Omron CX-Programmer project NewProject (CX-Programmer 9.61)

# PLC NewPLC1: CJ2M CPU31
I/O table (CPU CJ2M-CPU31): rack 0 slot 0 CJ1W-AD041-V1; rack 0 slot 1 CJ1W-ID211; rack 0 slot 2 CJ1W-OD211; rack 0 slot 3 CJ1W-DA041; rack 0 slot 11 CJ2M-EIP21

## Global symbols (name address type ; comment)
0.00 BOOL  ; PB_EMERGENCY STOP
0.01 BOOL  ; PB_MAN/AUTO
0.02 BOOL  ; PB_START
0.03 BOOL  ; PB_STOP
0.04 BOOL  ; PB_RESET
0.05 BOOL  ; PART SENSOR
0.06 BOOL  ; JIG IAI RIGHT END
0.07 BOOL  ; JIG IAI LEFT END
0.08 BOOL  ; JIG IAI ALARM
0.09 BOOL  ; INKJET IAI UP END
0.10 BOOL  ; INKJET IAI DOWN END
0.11 BOOL  ; INKJET IAI ALARM
0.12 BOOL  ; INKJET ERROR
0.13 BOOL  ; INKJET REFILL WARNING
0.14 BOOL  ; INKJET READY
0.15 BOOL  ; SPARE
1519.11 BOOL  ; Sequence end complete
1519.15 BOOL  ; Protocol Macro Executing
1.00 BOOL  ; LAMP PB_START
1.01 BOOL  ; JIG IAI RIGHT
1.02 BOOL  ; JIG IAI LEFT
1.03 BOOL  ; INKJET IAI UP
1.04 BOOL  ; INKJET IAI DOWN
1.05 BOOL  ; ALL IAI RESET ALARM
1.06 BOOL  ; BUZZER
1.07 BOOL  ; TWL YELLOW
1.08 BOOL  ; TWL GREEN
1.09 BOOL  ; TWL RED
1.10 BOOL  ; GREEN OK TWL
1.11 BOOL  ; RED NG TWL
2.00 BOOL  ; INKJET X4 IN1
2.01 BOOL  ; INKJET X4 IN2
2.02 BOOL  ; INKJET X4 IN3
2.03 BOOL  ; INKJET X4 JOB0
2.04 BOOL  ; INKJET X4 JOB1
2.05 BOOL  ; INKJET X4 JOB2
2.06 BOOL  ; INKJET X4 JOB3
2.07 BOOL  ; INKJET X4 JOB4
2.08 BOOL  ; INKJET X4 JOB5
2.09 BOOL  ; INKJET X4 JOB6
2.10 BOOL  ; INKJET X4 JOB7
2.11 BOOL  ; PRINT GO
3.00 BOOL  ; SOL ROTATE WORKPIECE ADV.
3.01 BOOL  ; SOL ROTATE WORKPIECE RET.
3.02 BOOL  ; SOL EJECTOR WORK NG ADV.
3.03 BOOL  ; SOL EJECTOR WORK NG RET.
3.04 BOOL  ; SOL CUT-OFF ADV.
3.05 BOOL  ; SOL CUT-OFF RET.
3.06 BOOL  ; SOL HOPPER ADV.
3.07 BOOL  ; SOL HOPPER RET.
3.08 BOOL  ; + JOB SELECT 0 (INKJET)
3.09 BOOL  ; + JOB SELECT 1 (INKJET)
3.10 BOOL  ; + JOB SELECT 2 (INKJET)
3.11 BOOL  ; + JOB SELECT 3 (INKJET)
3.12 BOOL  ; + JOB SELECT 4 (INKJET)
3.13 BOOL  ; + JOB SELECT 5 (INKJET)
3.14 BOOL  ; + JOB SELECT 6 (INKJET)
3.15 BOOL  ; + JOB SELECT 7 (INKJET)
40.09 BOOL  ; WARNING PRINT AGAIN
500.00 BOOL  ; SR-1000_PLC timming area
700.02 BOOL  ; TS170 TP WRITE DATA
750.05 BOOL  ; READING OK SV
850.00 BOOL  ; B-15 MANUAL HOME SELECT
950.00 BOOL  ; DTAT LOG INPUT
A202.07 BOOL  ; Com port Enable
A280.03 BOOL  ; COMPLETE
A280.05 BOOL  ; SERVO HOME
D0 CHANNEL  ; SCREEN CHANGE
D1 CHANNEL  ; 50.0% vari to G3PW
D100 CHANNEL  ; COUNTER PART
D1000 CHANNEL  ; MODEL NAME RUNNING
D102 CHANNEL  ; COUNTER PART NG
D1030 CHANNEL  ; PARM Q'TY BOX
D1050.00 BOOL  ; + JOB SELECT 0 (PLC PARAMETER)
D1050.01 BOOL  ; + JOB SELECT 1 (PLC PARAMETER)
D1050.02 BOOL  ; + JOB SELECT 2 (PLC PARAMETER)
D1050.03 BOOL  ; + JOB SELECT 3 (PLC PARAMETER)
D1050.04 BOOL  ; + JOB SELECT 4 (PLC PARAMETER)
D1050.05 BOOL  ; + JOB SELECT 5 (PLC PARAMETER)
D1050.06 BOOL  ; + JOB SELECT 6 (PLC PARAMETER)
D1050.07 BOOL  ; + JOB SELECT 7 (PLC PARAMETER)
D107 CHANNEL  ; DELAY BEFORE ADV
D108 CHANNEL  ; STATE OK NG
D110 CHANNEL  ; CYCLE TIME
D112 CHANNEL  ; CYCLE TIME
D114 CHANNEL  ; BARCODE TRIG DELAY
D116 CHANNEL  ; EJECTOR DELAY
D15 CHANNEL  ; TSC SET DELAY START
D19 CHANNEL  ; STATUS DISPLAY
D1900 CHANNEL  ; MODEL 1Y  2Wh 3BL 4Grey
D196 CHANNEL  ; CHANGE BOX NUMBER.
D1990 CHANNEL  ; MODEL NUMBER
D200 CHANNEL  ; FLT OKPART COUNT
D2000 CHANNEL  ; SCANNER DATA COMPARE
D210 CHANNEL  ; FEEDRATE COUNT
D220 CHANNEL  ; Password
D230 CHANNEL  ; FEERATE TSC.
D232 CHANNEL  ; OK PART COUNT
D234 CHANNEL  ; CHANGE BOX COUNT.
D236 CHANNEL  ; AGV SHOT TARGET
D240 CHANNEL  ; PART/SHOT COUNT
D244 CHANNEL  ; NG COUNT ALARM
D246 CHANNEL  ; NG COUNT TARGET
D248 CHANNEL  ; TIME OUT ALARM
D2500 CHANNEL  ; Cear Events Password
D260 CHANNEL  ; SHOT COUNT
D30000 CHANNEL  ; DATALOGGING
D3001.01 BOOL  ; ok
D3001.02 BOOL  ; ng
D3002.00 BOOL  ; Fins Ok
D3002.01 BOOL  ; Cam ok
D400 CHANNEL  ; DATA READ FROM SCANNER
D4990 CHANNEL  ; MODEL NUMBER
D4992 CHANNEL  ; MODEL NUMBER -1
D4994 CHANNEL  ; MODEL NUMBER -1*200
D4996 CHANNEL  ; ADDRESS START
D5000 CHANNEL  ; PARAMETER MODEL NAME
D504 CHANNEL  ; DATA READ FROM SCANNER
D600 CHANNEL  ; DATA READ FROM SCANNER IN PAGE32
D810 CHANNEL  ; POSITION FORM SELECT
D900 CHANNEL  ; AUTO DATA READ FROMSCANNER
H0.01 BOOL  ; MANUAL SELECT
H0.02 BOOL  ; AUTO SELECT
H100.00 BOOL  ; Z SELECT DIRECTION
H10.00 BOOL  ; STATE SIZE 80 USED
H10.01 BOOL  ; STATE SIZE 100 USE
H10.02 BOOL  ; STATE SIZE 150 USED
H11.00 BOOL  ; SIZE 80 USED
H11.01 BOOL  ; SIZE 100 USED
H11.02 BOOL  ; SIZE 150 USED
H12 CHANNEL  ; CHANGE PIC MODEL
H25.00 BOOL  ; USE COLOR DETECT
H420.15 BOOL  ; ALL FAULT(OFF)
H7.00 BOOL  ; SWITCH SELECTED
H7.01 BOOL  ; SENSOR SELECTED
H8.00 BOOL  ; BARCODE DISABLE
H8.01 BOOL  ; USE/UN USE INKJET
H8.02 BOOL  ; CHANGE BOX.
T0000 BOOL  ; BEFORE FLIP CYL. ADV
T0001 BOOL  ; AFTER FLIP CYL. ADV
T0008 BOOL  ; SS MODE MANUAL/AUTO [0.04] On
T0009 BOOL  ; SS MODE MANUAL/AUTO [0.04] Off
T0020 BOOL  ; DELAY START FROM SENSOR
T0021 BOOL  ; POWER ON TIME
T0050 BOOL  ; DELAY START BOWL
T0051 BOOL  ; DELAY PRINT GO
T0055 BOOL  ; NG BUFFER1 RUNNING
T0056 BOOL  ; NG BUFFER2 RUNNING
T0070 BOOL  ; EJECTOR TRIG BUFFER1
T0073 BOOL  ; EJECTOR TRIG BUFFER2
T0081 BOOL  ; EJECTOR RIGHT ALM.
T0082 BOOL  ; BUFFER BOX ADV. ALM.
T0083 BOOL  ; BUFFER BOX RET ALM.
T0092 BOOL  ; TIME OFF NG
T0093 BOOL  ; TIME OUT
T0098 BOOL  ; READ DONE
T0100 BOOL  ; AS EJECTOR WORK NG ADV. [1.02] On
T0101 BOOL  ; AS EJECTOR WORK NG RET. [1.03] On
T0102 BOOL  ; NG BUFFER3 RUNNING
T0103 BOOL  ; AS CUT-OFF RET. [1.05] On
T0104 BOOL  ; AS HOPPER ADV. [1.06] On
T0105 BOOL  ; AS HOPPER RET. [1.07] On
T0110 BOOL  ; AS ROTATE WORK PIECE ADV. [1.00] On
T0111 BOOL  ; AS ROTATE WORK PIECE RET. [1.01] On
T0152 BOOL  ; PH CHECK WORK EJECTOR  [1.10] On
T0153 BOOL  ; PH CHECK WORK EJECTOR  [1.10] Off
T0155 BOOL  ; PH CHECK WORK COUNTER [1.11] Off
T1002 BOOL  ; TIMER PREPARE DATA
T2000 BOOL  ; TIMER MODEL NAME SET
W0.00 BOOL  ; EMERGENCY STOP PB.
W0.01 BOOL  ; MANUAL MODE
W0.02 BOOL  ; AUTO MODE
W0.03 BOOL  ; MANUAL MODE PB. TSC.
W0.04 BOOL  ; AUTO MODE PB. TSC.
W0.10 BOOL  ; SET FLIP CYL ADV.
W100.00 BOOL  ; PB_EMERGENCY STOP
W100.01 BOOL  ; PB_MAN/AUTO
W100.02 BOOL  ; PB_START
W100.03 BOOL  ; PB_STOP
W100.04 BOOL  ; PB_RESET
W100.05 BOOL  ; PART SENSOR
W100.06 BOOL  ; JIG IAI RIGHT END
W100.07 BOOL  ; JIG IAI LEFT END
W100.08 BOOL  ; JIG IAI ALARM
W100.09 BOOL  ; INKJET IAI UP END
W100.10 BOOL  ; INKJET IAI DOWN END
W100.11 BOOL  ; INKJET IAI ALARM
W100.12 BOOL  ; INKJET ERROR
W100.13 BOOL  ; INKJET REFILL WARNING
W100.14 BOOL  ; INKJET READY
W100.15 BOOL  ; SPARE
W101.00 BOOL  ; LAMP PB_START
W101.01 BOOL  ; JIG IAI RIGHT
W101.02 BOOL  ; JIG IAI LEFT
W101.03 BOOL  ; INKJET IAI UP
W101.04 BOOL  ; INKJET IAI DOWN
W101.05 BOOL  ; ALL IAI RESET ALARM
W101.06 BOOL  ; INKJET PRINT GO
W101.07 BOOL  ; INKJET X4 IN1
W101.08 BOOL  ; INKJET X4 IN2
W101.09 BOOL  ; INKJET X4 IN2
W101.10 BOOL  ; INKJET X4 JOB0
W101.11 BOOL  ; INKJET X4 JOB1
W101.12 BOOL  ; INKJET X4 JOB2
W101.13 BOOL  ; TWL YELLOW
W101.14 BOOL  ; TWL GREEN
W101.15 BOOL  ; TWL RED
W102.00 BOOL  ; GREEN OK TWL
W102.01 BOOL  ; RED NG TWL
W10.00 BOOL  ; A/JIG IAI RIGHT
W10.01 BOOL  ; A/JIG IAI LEFT
W10.02 BOOL  ; A/INKJET IAI UP
W10.03 BOOL  ; A/INKJET IAI DOWN
W10.04 BOOL  ; A/CONVEYOR START
W10.05 BOOL  ; A/BOWL START
W10.06 BOOL  ; A/PRINT GO
W10.07 BOOL  ; NG BUFFER1
W10.08 BOOL  ; NG BUFFER2
W10.09 BOOL  ; SET NG BUFFER1
W10.10 BOOL  ; SET NG BUFFER2
W10.11 BOOL  ; SET NG BUFFER3
W10.12 BOOL  ; NG BUFFER3
W10.13 BOOL  ; A/SHOT TRIG TO AGV
W10.15 BOOL  ; HOME
W11.00 BOOL  ; EJECTOR RUNNING
W11.01 BOOL  ; CALL JOB 0
W11.02 BOOL  ; CALL JOB 1
W11.03 BOOL  ; CALL JOB 2
W13.00 BOOL  ; CALL JOB 0
W13.01 BOOL  ; CALL JOB 1
W13.02 BOOL  ; CALL JOB 2
W15.00 BOOL  ; BIT TRIG SHOT
W15.01 BOOL  ; AGV LOADING START COUNT BUFFER
W1.00 BOOL  ; start communication
W1.01 BOOL  ; CYCLE START
W1.02 BOOL  ; RETURN DONE
W1.03 BOOL  ; MACHINE READY
W1.04 BOOL  ; A/PRINT GO(DOWN)
W1.05 BOOL  ; A/PRINT GO(UP)
W1.13 BOOL  ; TEST LAMP
W200.11 BOOL  ; AUTO RUNNING
W202.10 BOOL  ; BARCODE CHECK OK
W202.11 BOOL  ; BARCODE CHECK NG
W204.02 BOOL  ; EJECT WORK RUNNING
W20.00 BOOL  ; Delay Check Barcode
W21.00 BOOL  ; ROBOT STOP
W25.02 BOOL  ; FLAG TO DECRETE NG
W26.03 BOOL  ; GREEN
W26.05 BOOL  ; RED
W300.00 BOOL  ; TRIG COLOR DETECT
W300.01 BOOL  ; FINS OK
W300.02 BOOL  ; CAM CONNECT
W300.03 BOOL  ; DETECT OK
W300.04 BOOL  ; DETECT NG
W302.00 BOOL  ; RECORD Y
W302.01 BOOL  ; RECORD WH
W303.00 BOOL  ; MAN. READ COLOR
W304.00 BOOL  ; WARNING CORLOR DETECTION
W305.00 BOOL  ; FIRST START CHECK COLOR
W30.00 BOOL  ; TRIG HMI MACRO 00
W30.01 BOOL  ; TRIG MACRO
W30.02 BOOL  ; TRIG MACRO AUTO PAGE
W345.00 BOOL  ; TS069 PB CLEAR BOX
W345.01 BOOL  ; TSC CLEAR POPUP
W345.02 BOOL  ; ENABLE JUDGMENT
W35 CHANNEL  ; INDIREC SCR AUTO PAGE
W350.00 BOOL  ; TSPL EJECTOR WORK NG ADV.
W350.01 BOOL  ; TSPL EJECTOR WORK NG RET.
W350.02 BOOL  ; TSPL CUT-OFF ADV.
W350.03 BOOL  ; TSPL CUT-OFF RET.
W350.04 BOOL  ; TSPL HOPPER ADV.
W350.05 BOOL  ; TSPL HOPPER RET.
W350.07 BOOL  ; TS PL SCANNER TRIG
W350.08 BOOL  ; TSPL MOTOR CONVEYOR ON
W350.09 BOOL  ; TSPL MOTOR CONVEYOR OFF
W350.10 BOOL  ; TSPL HOPPER BOWL FEEDER ON
W350.11 BOOL  ; TSPL HOPPER BOWL FEEDER OFF
W350.12 BOOL  ; TSPL BOWL FEEDER ON
W350.13 BOOL  ; TSPL BOWL FEEDER OFF
W350.14 BOOL  ; TSPL LINEAR BOWL FEEDER ON
W350.15 BOOL  ; TSPL LINEAR BOWL FEEDER OFF
W351.00 BOOL  ; TS PL ROTATE WORK PIECE ADV.
W351.01 BOOL  ; TS PL ROTATE WORK PIECE RET.
W36 CHANNEL  ; 400X250 INDIRECT SCR AUTO PAGE
W39.09 BOOL  ; ALL ALARM
W39.10 BOOL  ; ALARM
W401 CHANNEL  ; CURRENT SCREEN
W402 CHANNEL  ; CHANGE SCREEN
W40.01 BOOL  ; EMERGENCY STOP
W40.02 BOOL  ; DEVICES NOT HOME
W40.03 BOOL  ; PLC ERROR
W40.04 BOOL  ; PLC LOW BATTERY
W40.05 BOOL  ; JIG IAI ALARM
W40.06 BOOL  ; INKJET IAI ALARM
W40.07 BOOL  ; INKJET ERROR
W40.08 BOOL  ; INKJET REFILL WARNING
W40.09 BOOL  ; FLIP ROD RET. ALM
W40.10 BOOL  ; NG COUNT ALM.
W40.11 BOOL  ; OVER CYCLE TIME ALM.
W40.12 BOOL  ; DOOR OPENED
W40.13 BOOL  ; PART SENSOR ALM.
W40.14 BOOL  ; EJECTOR SENSOR ALM.
W40.15 BOOL  ; COUNTING SENSOR ALM.
W41.01 BOOL  ; CAM CONNECT ERROR
W41.02 BOOL  ; COLOR NOT DETECT
W42.00 BOOL  ; WARNING PRINT AGAIN
W442.00 BOOL  ; SW. ENTER PASSWORD
W442.15 BOOL  ; Unlock Cear Event Password
W459.00 BOOL  ; MACHINE READY
W45.00 BOOL  ; MACRO DETECT BARCODE DONE
W4.04 BOOL  ; ALL HOME START RUNNING
W500.00 BOOL  ; TS_PB READ
W500.01 BOOL  ; TS_PL READ
W500.02 BOOL  ; TS_PB SAVE
W500.03 BOOL  ; TS_PL SAVE
W500.04 BOOL  ; SAVE COMPLETE
W500.06 BOOL  ; INPUT MODEL CODE ITL.
W500.08 BOOL  ; SAVE RFID
W500.10 BOOL  ; READ COMPLETE
W500.12 BOOL  ; SAVE COMPLETE
W500.15 BOOL  ; PARM SETTING COND.
W501.00 BOOL  ; TS_PB SELLECT MODEL
W50.01 BOOL  ; UPLOAD DATA
W50.02 BOOL  ; PART COUNTER TARGET
W50.04 BOOL  ; Password OK
W55.00 BOOL  ; INKJET IAI UP
W55.01 BOOL  ; INKJET IAI DOWN
W55.02 BOOL  ; JIG IAI LEFT
W55.03 BOOL  ; JIG IAI RIGHT
W55.04 BOOL  ; CONVEYOR RUN
W55.05 BOOL  ; BOWL FEEDER START
W60.01 BOOL  ; PART TRIG BUFFER 1
W60.02 BOOL  ; SENSOR PART TRIG BUFFER1
W60.03 BOOL  ; SENSOR PART TRIG BUFFER2
W60.04 BOOL  ; PART TRIG BUFFER 2
W60.05 BOOL  ; PART TRIG BUFFER 3
W60.06 BOOL  ; BARCODE TRIG BUFFER1
W60.07 BOOL  ; BARCODE TRIG BUFFER2
W60.08 BOOL  ; BARCODE TRIG BUFFER3
W60.09 BOOL  ; EJECTOR PART TRIG BUFFER1
W60.10 BOOL  ; EJECTOR PART TRIG BUFFER2
W60.11 BOOL  ; EJECTOR PART TRIG BUFFER3
W61.00 BOOL  ; SENSOR PART TRIG BUFFER3
W62.01 BOOL  ; START FROM ROBOT
W63.00 BOOL  ; TSC STATE STOP
W63.01 BOOL  ; TSC BOWL STATE STOP
W64.00 BOOL  ; M/TSC JIG IAI RIGHT
W64.01 BOOL  ; M/TSC JIG IAI LEFT
W64.02 BOOL  ; M/TSC INKJET IAI UP
W64.03 BOOL  ; M/TSC INKJET IAI DOWN
W64.04 BOOL  ; M/TSC BUFFER BOX ADV
W64.05 BOOL  ; M/TSC BUFFER BOX RET
W64.06 BOOL  ; M/TSC BELT START
W64.07 BOOL  ; M/TSC BELT STOP
W64.08 BOOL  ; M/TSC BOWL START
W64.09 BOOL  ; M/TSC BOWL STOP
W64.15 BOOL  ; barcode trigger
W65.00 BOOL  ; A/BARCODE TRIG
W65.14 BOOL  ; MAN/CLEAR BARCODE
W65.15 BOOL  ; TEST TRIGGER
W69.00 BOOL  ; P E A R
W6.06 BOOL  ; PUASE TO TSC
W6.07 BOOL  ; TSC CLEAR OK
W6.08 BOOL  ; TSC CLEAR COUNT
W6.09 BOOL  ; ALARM RESET
W6.10 BOOL  ; ALARM DISPLAY
W6.11 BOOL  ; ALL HOME
W6.12 BOOL  ; HOME TSC.
W6.15 BOOL  ; CLEAR SHOT
W70.00 BOOL  ; PART TRIG BUFFER 4
W70.01 BOOL  ; PART TRIG BUFFER 5
W70.02 BOOL  ; BARCODE TRIG BUFFER4
W70.03 BOOL  ; BARCODE TRIG BUFFER5
W71.00 BOOL  ; SENSOR PART TRIG TO CLEAR
W7.00 BOOL  ; TSC SWITCH SELECT
W7.01 BOOL  ; TSC SENSOR SELECT
W7.05 BOOL  ; PROTECT PRINT AGAIN
W80.00 BOOL  ; H.BARCODE OK
W80.01 BOOL  ; H.BARCODE NG
W8.01 BOOL  ; COUNT DONE
W8.02 BOOL  ; A/BUFFER BOX RELEASE
W8.03 BOOL  ; CHANGE BOX OK.
W8.04 BOOL  ; TSC CLEAR NG
W8.09 BOOL  ; AGV LOADING
W90.00 BOOL  ; OK
W90.01 BOOL  ; OK
W90.02 BOOL  ; NG
W90.03 BOOL  ; NG
W90.14 BOOL  ; SETTING
W90.15 BOOL  ; READ COMPLETE
W91.00 BOOL  ; CREATE BARCODE 80
W91.01 BOOL  ; CREATE BARCODE 100
W91.02 BOOL  ; CREATE BARCODE 150

## Program NewProgram1 (cyclic task 0)
Local symbols
P_On CF113 BOOL
Ğ98 BOOL

### Section ScreenOperation

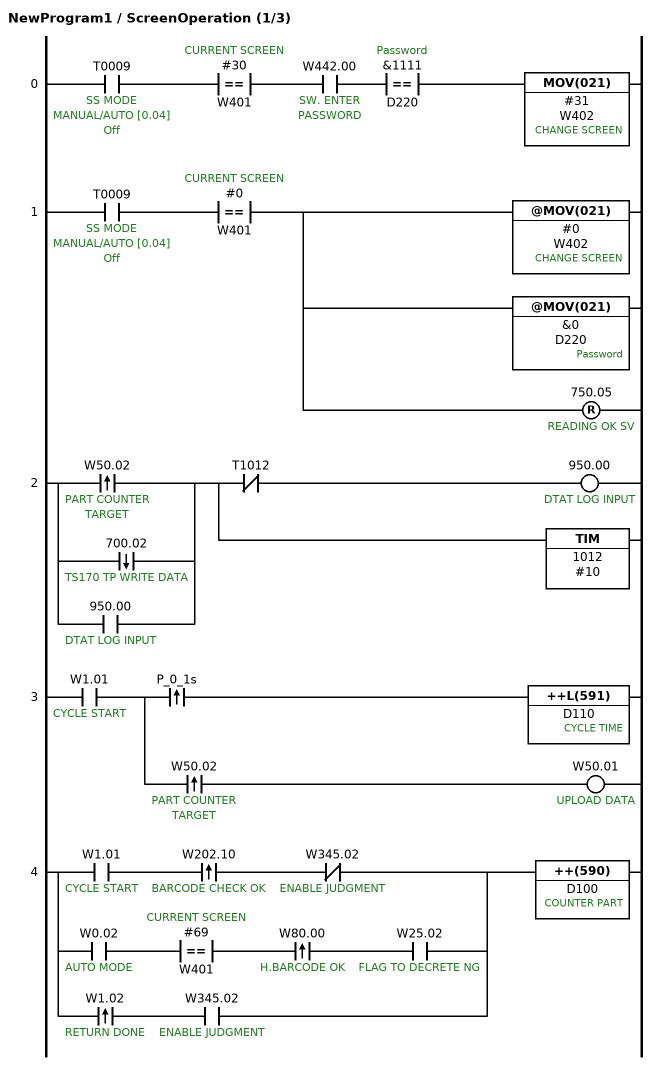
; rung 0
LD T0009  ; SS MODE MANUAL/AUTO [0.04] Off
AND=(300) #30 W401  ; CURRENT SCREEN
AND W442.00  ; SW. ENTER PASSWORD
AND=(300) &1111 D220  ; Password
MOV(021) #31 W402  ; CHANGE SCREEN
; rung 1
LD T0009  ; SS MODE MANUAL/AUTO [0.04] Off
AND=(300) #0 W401  ; CURRENT SCREEN
@MOV(021) #0 W402  ; CHANGE SCREEN
@MOV(021) &0 D220  ; Password
RSET 750.05  ; READING OK SV
; rung 2
@LD W50.02  ; PART COUNTER TARGET
%OR 700.02  ; TS170 TP WRITE DATA
OR 950.00  ; DTAT LOG INPUT
OUT TR0
ANDNOT T1012
OUT 950.00  ; DTAT LOG INPUT
LD TR0
TIM 1012 #10
; rung 3
LD W1.01  ; CYCLE START
OUT TR0
@AND P_0_1s
++L(591) D110  ; CYCLE TIME
LD TR0
@AND W50.02  ; PART COUNTER TARGET
OUT W50.01  ; UPLOAD DATA
; rung 4
LD W1.01  ; CYCLE START
@AND W202.10  ; BARCODE CHECK OK
ANDNOT W345.02  ; ENABLE JUDGMENT
LD W0.02  ; AUTO MODE
AND=(300) #69 W401  ; CURRENT SCREEN
@AND W80.00  ; H.BARCODE OK
AND W25.02  ; FLAG TO DECRETE NG
ORLD
@LD W1.02  ; RETURN DONE
AND W345.02  ; ENABLE JUDGMENT
ORLD
++(590) D100  ; COUNTER PART

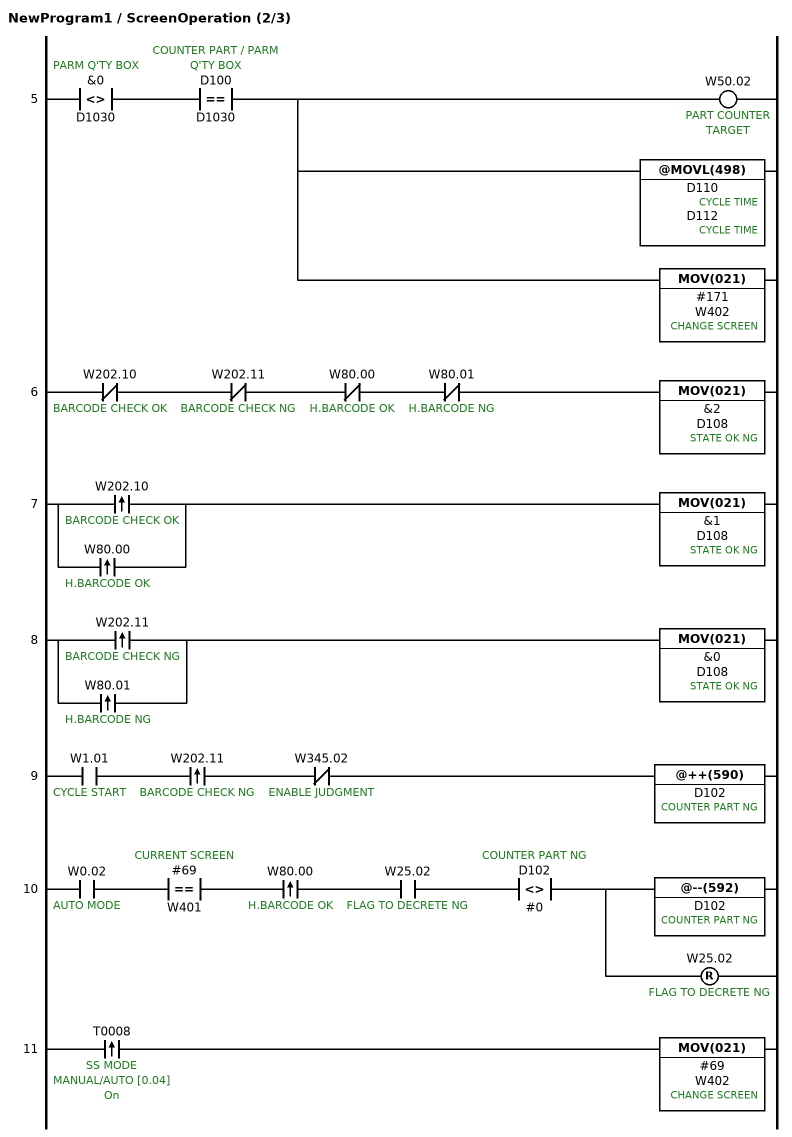
; rung 5
LD<>(305) &0 D1030  ; PARM Q'TY BOX
AND=(300) D100 D1030  ; COUNTER PART, PARM Q'TY BOX
OUT W50.02  ; PART COUNTER TARGET
@MOVL(498) D110 D112  ; CYCLE TIME
MOV(021) #171 W402  ; CHANGE SCREEN
; rung 6
LDNOT W202.10  ; BARCODE CHECK OK
ANDNOT W202.11  ; BARCODE CHECK NG
ANDNOT W80.00  ; H.BARCODE OK
ANDNOT W80.01  ; H.BARCODE NG
MOV(021) &2 D108  ; STATE OK NG
; rung 7
@LD W202.10  ; BARCODE CHECK OK
@OR W80.00  ; H.BARCODE OK
MOV(021) &1 D108  ; STATE OK NG
; rung 8
@LD W202.11  ; BARCODE CHECK NG
@OR W80.01  ; H.BARCODE NG
MOV(021) &0 D108  ; STATE OK NG
; rung 9
LD W1.01  ; CYCLE START
@AND W202.11  ; BARCODE CHECK NG
ANDNOT W345.02  ; ENABLE JUDGMENT
@++(590) D102  ; COUNTER PART NG
; rung 10
LD W0.02  ; AUTO MODE
AND=(300) #69 W401  ; CURRENT SCREEN
@AND W80.00  ; H.BARCODE OK
AND W25.02  ; FLAG TO DECRETE NG
AND<>(305) D102 #0  ; COUNTER PART NG
@--(592) D102  ; COUNTER PART NG
RSET W25.02  ; FLAG TO DECRETE NG
; rung 11
@LD T0008  ; SS MODE MANUAL/AUTO [0.04] On
MOV(021) #69 W402  ; CHANGE SCREEN

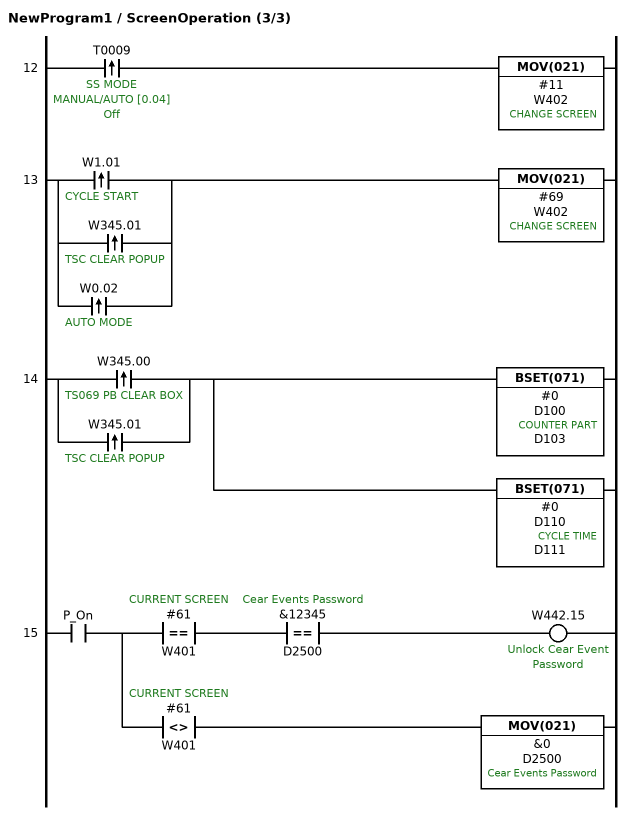
; rung 12
@LD T0009  ; SS MODE MANUAL/AUTO [0.04] Off
MOV(021) #11 W402  ; CHANGE SCREEN
; rung 13
@LD W1.01  ; CYCLE START
@OR W345.01  ; TSC CLEAR POPUP
@OR W0.02  ; AUTO MODE
MOV(021) #69 W402  ; CHANGE SCREEN
; rung 14
@LD W345.00  ; TS069 PB CLEAR BOX
@OR W345.01  ; TSC CLEAR POPUP
BSET(071) #0 D100 D103  ; COUNTER PART
BSET(071) #0 D110 D111  ; CYCLE TIME
; rung 15
LD P_On
OUT TR0
AND=(300) #61 W401  ; CURRENT SCREEN
AND=(300) &12345 D2500  ; Cear Events Password
OUT W442.15  ; Unlock Cear Event Password
LD TR0
AND<>(305) #61 W401  ; CURRENT SCREEN
MOV(021) &0 D2500  ; Cear Events Password

### Section MODEL_SELLECT

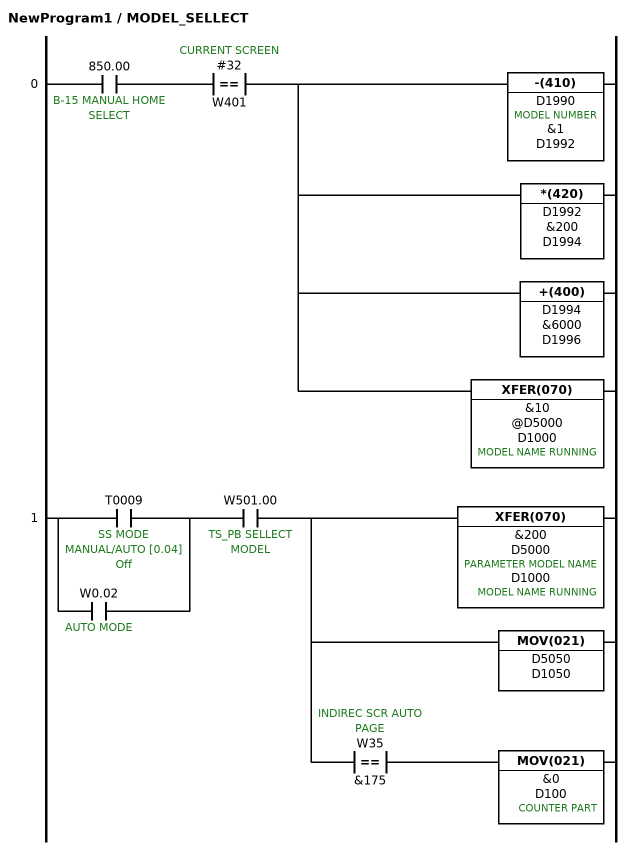
; rung 0
LD 850.00  ; B-15 MANUAL HOME SELECT
AND=(300) #32 W401  ; CURRENT SCREEN
-(410) D1990 &1 D1992  ; MODEL NUMBER
*(420) D1992 &200 D1994
+(400) D1994 &6000 D1996
XFER(070) &10 @D5000 D1000  ; MODEL NAME RUNNING
; rung 1
LD T0009  ; SS MODE MANUAL/AUTO [0.04] Off
OR W0.02  ; AUTO MODE
AND W501.00  ; TS_PB SELLECT MODEL
XFER(070) &200 D5000 D1000  ; PARAMETER MODEL NAME, MODEL NAME RUNNING
MOV(021) D5050 D1050
AND=(300) W35 &175  ; INDIREC SCR AUTO PAGE
MOV(021) &0 D100  ; COUNTER PART

### Section MODEL_SETING

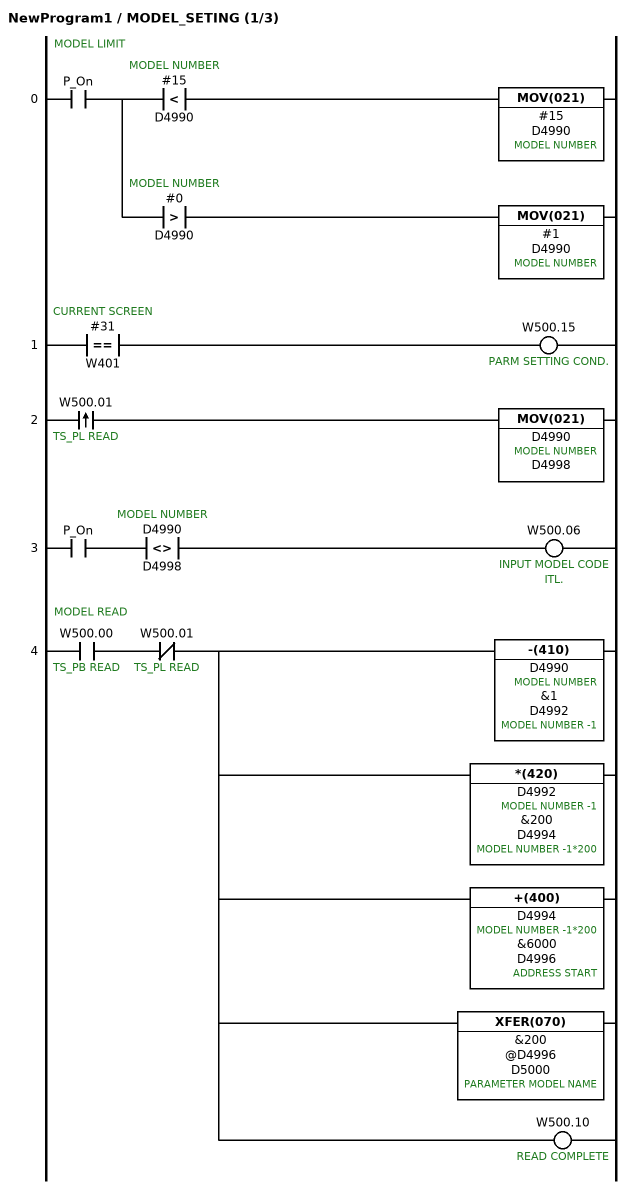
; rung 0: MODEL LIMIT
LD P_On
OUT TR0
AND<(310) #15 D4990  ; MODEL NUMBER
MOV(021) #15 D4990  ; MODEL NUMBER
LD TR0
AND>(320) #0 D4990  ; MODEL NUMBER
MOV(021) #1 D4990  ; MODEL NUMBER
; rung 1
LD=(300) #31 W401  ; CURRENT SCREEN
OUT W500.15  ; PARM SETTING COND.
; rung 2
@LD W500.01  ; TS_PL READ
MOV(021) D4990 D4998  ; MODEL NUMBER
; rung 3
LD P_On
AND<>(305) D4990 D4998  ; MODEL NUMBER
OUT W500.06  ; INPUT MODEL CODE ITL.
; rung 4: MODEL READ
LD W500.00  ; TS_PB READ
ANDNOT W500.01  ; TS_PL READ
-(410) D4990 &1 D4992  ; MODEL NUMBER, MODEL NUMBER -1
*(420) D4992 &200 D4994  ; MODEL NUMBER -1, MODEL NUMBER -1*200
+(400) D4994 &6000 D4996  ; MODEL NUMBER -1*200, ADDRESS START
XFER(070) &200 @D4996 D5000  ; PARAMETER MODEL NAME
OUT W500.10  ; READ COMPLETE

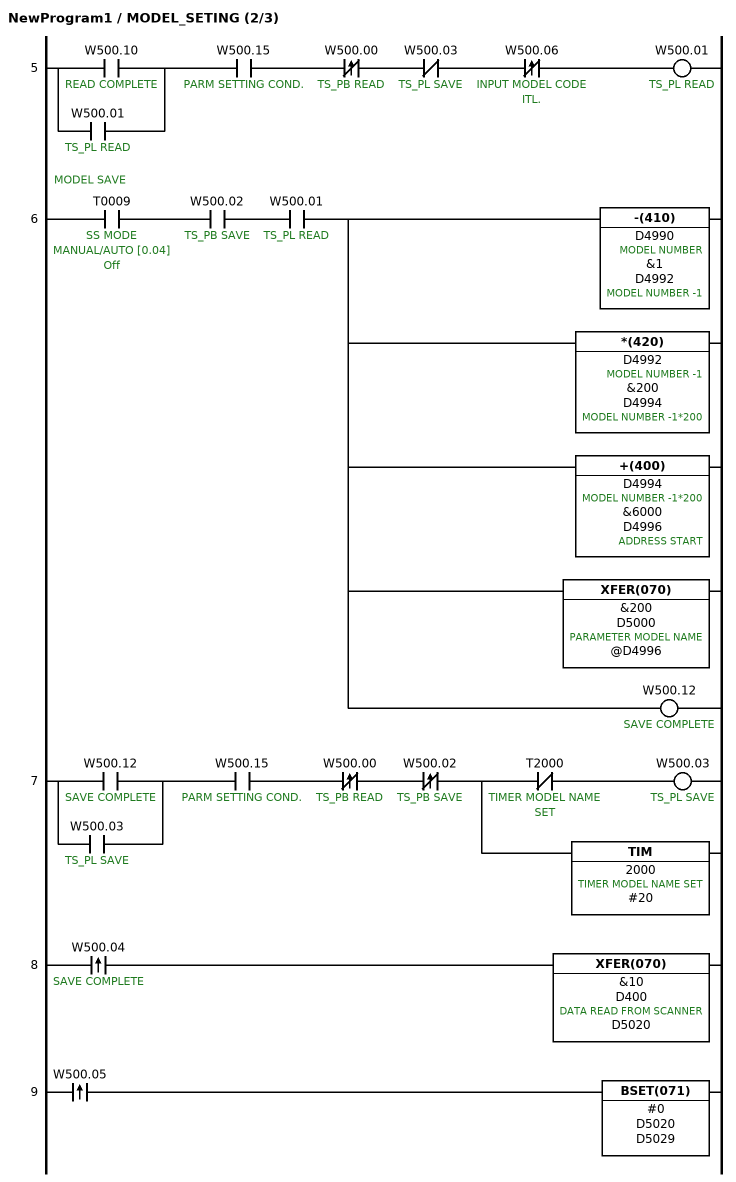
; rung 5
LD W500.10  ; READ COMPLETE
OR W500.01  ; TS_PL READ
AND W500.15  ; PARM SETTING COND.
@ANDNOT W500.00  ; TS_PB READ
ANDNOT W500.03  ; TS_PL SAVE
@ANDNOT W500.06  ; INPUT MODEL CODE ITL.
OUT W500.01  ; TS_PL READ
; rung 6: MODEL SAVE
LD T0009  ; SS MODE MANUAL/AUTO [0.04] Off
AND W500.02  ; TS_PB SAVE
AND W500.01  ; TS_PL READ
-(410) D4990 &1 D4992  ; MODEL NUMBER, MODEL NUMBER -1
*(420) D4992 &200 D4994  ; MODEL NUMBER -1, MODEL NUMBER -1*200
+(400) D4994 &6000 D4996  ; MODEL NUMBER -1*200, ADDRESS START
XFER(070) &200 D5000 @D4996  ; PARAMETER MODEL NAME
OUT W500.12  ; SAVE COMPLETE
; rung 7
LD W500.12  ; SAVE COMPLETE
OR W500.03  ; TS_PL SAVE
AND W500.15  ; PARM SETTING COND.
@ANDNOT W500.00  ; TS_PB READ
@ANDNOT W500.02  ; TS_PB SAVE
OUT TR0
ANDNOT T2000  ; TIMER MODEL NAME SET
OUT W500.03  ; TS_PL SAVE
LD TR0
TIM 2000 #20  ; TIMER MODEL NAME SET
; rung 8
@LD W500.04  ; SAVE COMPLETE
XFER(070) &10 D400 D5020  ; DATA READ FROM SCANNER
; rung 9
@LD W500.05
BSET(071) #0 D5020 D5029

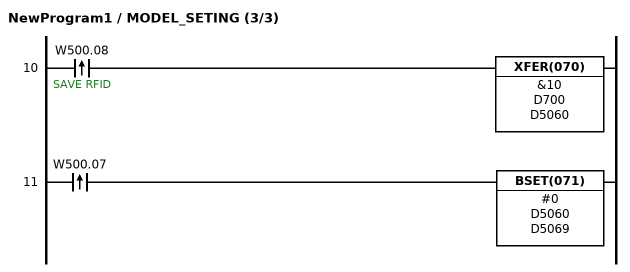
; rung 10
@LD W500.08  ; SAVE RFID
XFER(070) &10 D700 D5060
; rung 11
@LD W500.07
BSET(071) #0 D5060 D5069

### Section MAIN

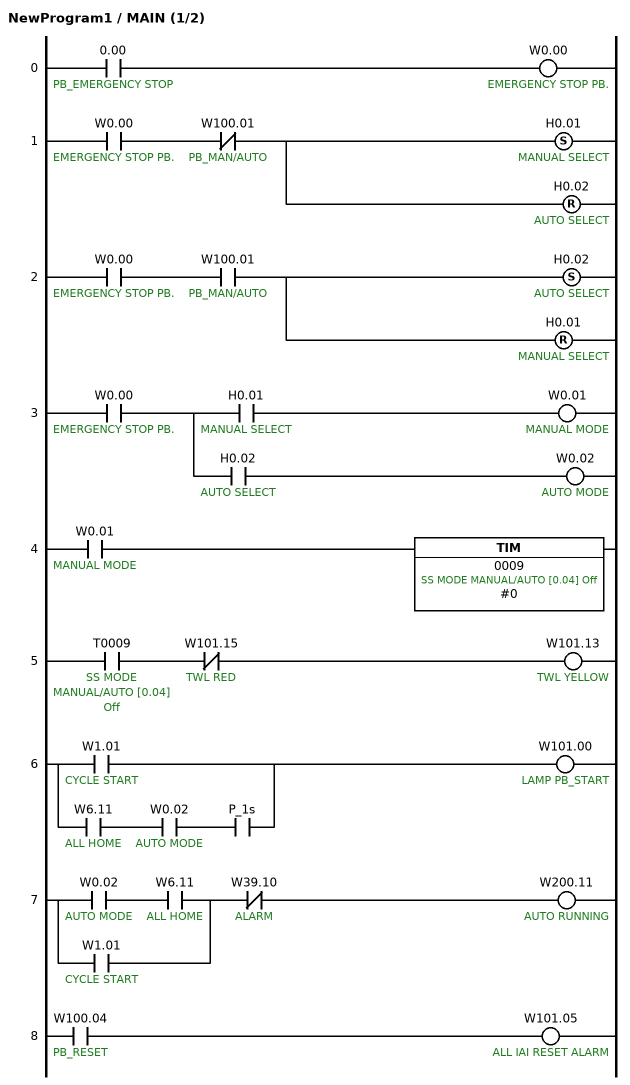
; rung 0
LD 0.00  ; PB_EMERGENCY STOP
OUT W0.00  ; EMERGENCY STOP PB.
; rung 1
LD W0.00  ; EMERGENCY STOP PB.
ANDNOT W100.01  ; PB_MAN/AUTO
SET H0.01  ; MANUAL SELECT
RSET H0.02  ; AUTO SELECT
; rung 2
LD W0.00  ; EMERGENCY STOP PB.
AND W100.01  ; PB_MAN/AUTO
SET H0.02  ; AUTO SELECT
RSET H0.01  ; MANUAL SELECT
; rung 3
LD W0.00  ; EMERGENCY STOP PB.
OUT TR0
AND H0.01  ; MANUAL SELECT
OUT W0.01  ; MANUAL MODE
LD TR0
AND H0.02  ; AUTO SELECT
OUT W0.02  ; AUTO MODE
; rung 4
LD W0.01  ; MANUAL MODE
TIM 0009 #0  ; SS MODE MANUAL/AUTO [0.04] Off
; rung 5
LD T0009  ; SS MODE MANUAL/AUTO [0.04] Off
ANDNOT W101.15  ; TWL RED
OUT W101.13  ; TWL YELLOW
; rung 6
LD W1.01  ; CYCLE START
LD W6.11  ; ALL HOME
AND W0.02  ; AUTO MODE
AND P_1s
ORLD
OUT W101.00  ; LAMP PB_START
; rung 7
LD W0.02  ; AUTO MODE
AND W6.11  ; ALL HOME
OR W1.01  ; CYCLE START
ANDNOT W39.10  ; ALARM
OUT W200.11  ; AUTO RUNNING
; rung 8
LD W100.04  ; PB_RESET
OUT W101.05  ; ALL IAI RESET ALARM

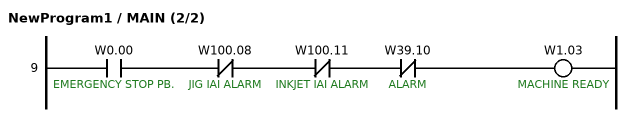
; rung 9
LD W0.00  ; EMERGENCY STOP PB.
ANDNOT W100.08  ; JIG IAI ALARM
ANDNOT W100.11  ; INKJET IAI ALARM
ANDNOT W39.10  ; ALARM
OUT W1.03  ; MACHINE READY

### Section AUTO

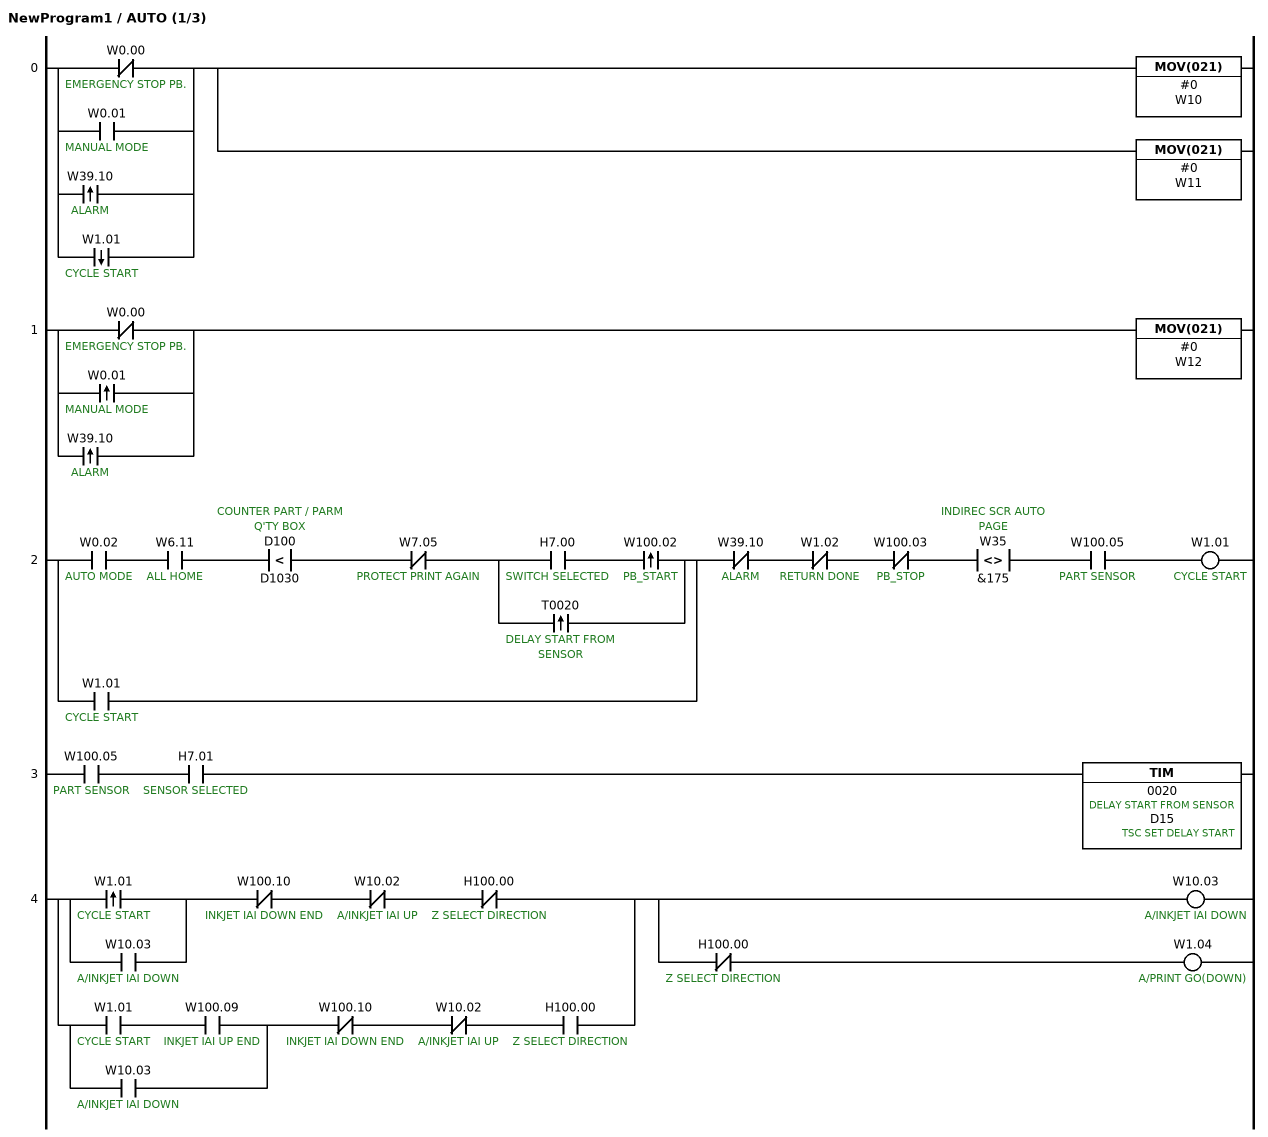
; rung 0
LDNOT W0.00  ; EMERGENCY STOP PB.
OR W0.01  ; MANUAL MODE
@OR W39.10  ; ALARM
%OR W1.01  ; CYCLE START
MOV(021) #0 W10
MOV(021) #0 W11
; rung 1
LDNOT W0.00  ; EMERGENCY STOP PB.
@OR W0.01  ; MANUAL MODE
@OR W39.10  ; ALARM
MOV(021) #0 W12
; rung 2
LD W0.02  ; AUTO MODE
AND W6.11  ; ALL HOME
AND<(310) D100 D1030  ; COUNTER PART, PARM Q'TY BOX
ANDNOT W7.05  ; PROTECT PRINT AGAIN
LD H7.00  ; SWITCH SELECTED
@AND W100.02  ; PB_START
@OR T0020  ; DELAY START FROM SENSOR
ANDLD
OR W1.01  ; CYCLE START
ANDNOT W39.10  ; ALARM
ANDNOT W1.02  ; RETURN DONE
ANDNOT W100.03  ; PB_STOP
AND<>(305) W35 &175  ; INDIREC SCR AUTO PAGE
AND W100.05  ; PART SENSOR
OUT W1.01  ; CYCLE START
; rung 3
LD W100.05  ; PART SENSOR
AND H7.01  ; SENSOR SELECTED
TIM 0020 D15  ; TSC SET DELAY START, DELAY START FROM SENSOR
; rung 4
@LD W1.01  ; CYCLE START
OR W10.03  ; A/INKJET IAI DOWN
ANDNOT W100.10  ; INKJET IAI DOWN END
ANDNOT W10.02  ; A/INKJET IAI UP
ANDNOT H100.00  ; Z SELECT DIRECTION
LD W1.01  ; CYCLE START
AND W100.09  ; INKJET IAI UP END
OR W10.03  ; A/INKJET IAI DOWN
ANDNOT W100.10  ; INKJET IAI DOWN END
ANDNOT W10.02  ; A/INKJET IAI UP
AND H100.00  ; Z SELECT DIRECTION
ORLD
OUT W10.03  ; A/INKJET IAI DOWN
ANDNOT H100.00  ; Z SELECT DIRECTION
OUT W1.04  ; A/PRINT GO(DOWN)

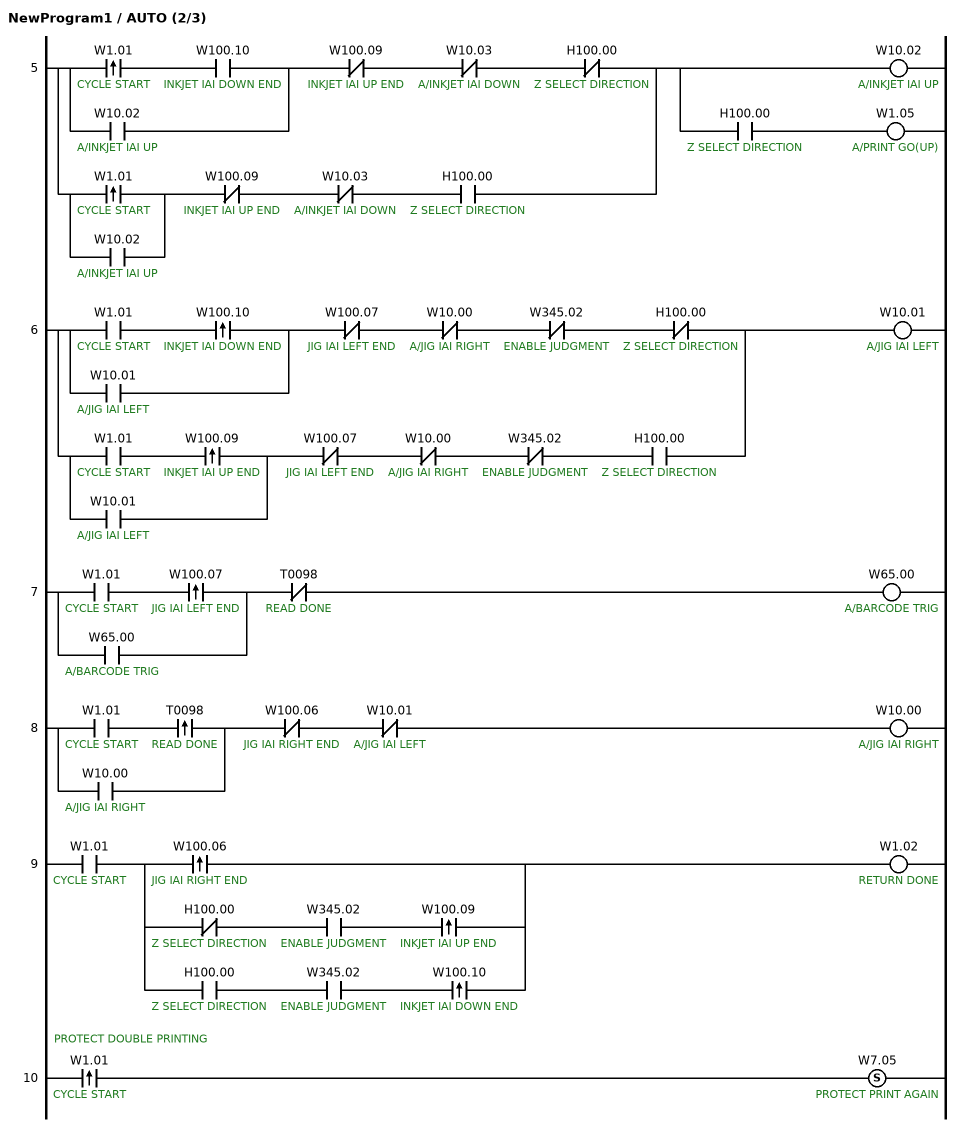
; rung 5
@LD W1.01  ; CYCLE START
AND W100.10  ; INKJET IAI DOWN END
OR W10.02  ; A/INKJET IAI UP
ANDNOT W100.09  ; INKJET IAI UP END
ANDNOT W10.03  ; A/INKJET IAI DOWN
ANDNOT H100.00  ; Z SELECT DIRECTION
@LD W1.01  ; CYCLE START
OR W10.02  ; A/INKJET IAI UP
ANDNOT W100.09  ; INKJET IAI UP END
ANDNOT W10.03  ; A/INKJET IAI DOWN
AND H100.00  ; Z SELECT DIRECTION
ORLD
OUT W10.02  ; A/INKJET IAI UP
AND H100.00  ; Z SELECT DIRECTION
OUT W1.05  ; A/PRINT GO(UP)
; rung 6
LD W1.01  ; CYCLE START
@AND W100.10  ; INKJET IAI DOWN END
OR W10.01  ; A/JIG IAI LEFT
ANDNOT W100.07  ; JIG IAI LEFT END
ANDNOT W10.00  ; A/JIG IAI RIGHT
ANDNOT W345.02  ; ENABLE JUDGMENT
ANDNOT H100.00  ; Z SELECT DIRECTION
LD W1.01  ; CYCLE START
@AND W100.09  ; INKJET IAI UP END
OR W10.01  ; A/JIG IAI LEFT
ANDNOT W100.07  ; JIG IAI LEFT END
ANDNOT W10.00  ; A/JIG IAI RIGHT
ANDNOT W345.02  ; ENABLE JUDGMENT
AND H100.00  ; Z SELECT DIRECTION
ORLD
OUT W10.01  ; A/JIG IAI LEFT
; rung 7
LD W1.01  ; CYCLE START
@AND W100.07  ; JIG IAI LEFT END
OR W65.00  ; A/BARCODE TRIG
ANDNOT T0098  ; READ DONE
OUT W65.00  ; A/BARCODE TRIG
; rung 8
LD W1.01  ; CYCLE START
@AND T0098  ; READ DONE
OR W10.00  ; A/JIG IAI RIGHT
ANDNOT W100.06  ; JIG IAI RIGHT END
ANDNOT W10.01  ; A/JIG IAI LEFT
OUT W10.00  ; A/JIG IAI RIGHT
; rung 9
LD W1.01  ; CYCLE START
@LD W100.06  ; JIG IAI RIGHT END
LDNOT H100.00  ; Z SELECT DIRECTION
AND W345.02  ; ENABLE JUDGMENT
@AND W100.09  ; INKJET IAI UP END
ORLD
LD H100.00  ; Z SELECT DIRECTION
AND W345.02  ; ENABLE JUDGMENT
@AND W100.10  ; INKJET IAI DOWN END
ORLD
ANDLD
OUT W1.02  ; RETURN DONE
; rung 10: PROTECT DOUBLE PRINTING
@LD W1.01  ; CYCLE START
SET W7.05  ; PROTECT PRINT AGAIN

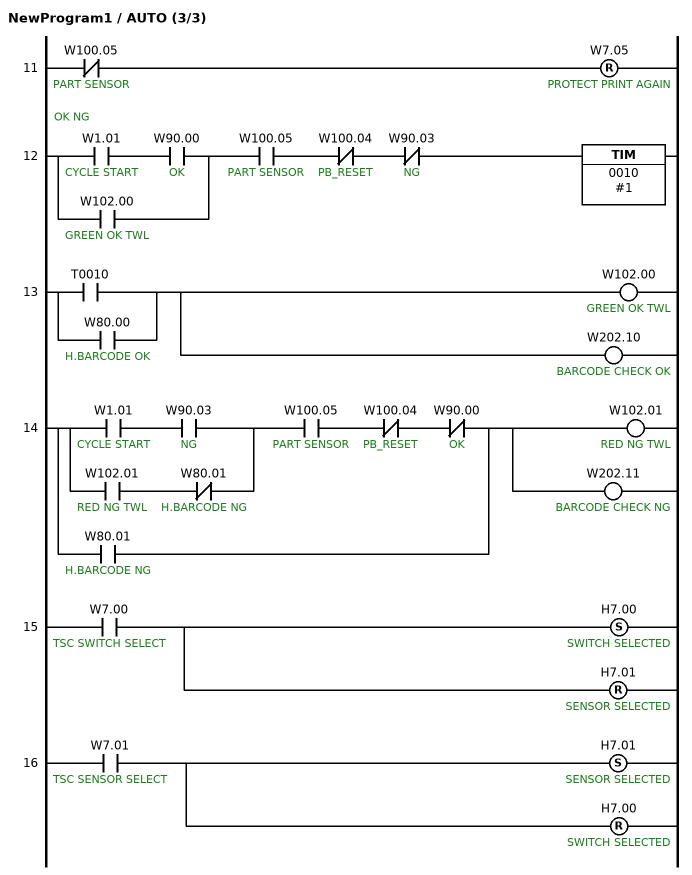
; rung 11
LDNOT W100.05  ; PART SENSOR
RSET W7.05  ; PROTECT PRINT AGAIN
; rung 12: OK NG
LD W1.01  ; CYCLE START
AND W90.00  ; OK
OR W102.00  ; GREEN OK TWL
AND W100.05  ; PART SENSOR
ANDNOT W100.04  ; PB_RESET
ANDNOT W90.03  ; NG
TIM 0010 #1
; rung 13
LD T0010
OR W80.00  ; H.BARCODE OK
OUT W102.00  ; GREEN OK TWL
OUT W202.10  ; BARCODE CHECK OK
; rung 14
LD W1.01  ; CYCLE START
AND W90.03  ; NG
LD W102.01  ; RED NG TWL
ANDNOT W80.01  ; H.BARCODE NG
ORLD
AND W100.05  ; PART SENSOR
ANDNOT W100.04  ; PB_RESET
ANDNOT W90.00  ; OK
OR W80.01  ; H.BARCODE NG
OUT W102.01  ; RED NG TWL
OUT W202.11  ; BARCODE CHECK NG
; rung 15
LD W7.00  ; TSC SWITCH SELECT
SET H7.00  ; SWITCH SELECTED
RSET H7.01  ; SENSOR SELECTED
; rung 16
LD W7.01  ; TSC SENSOR SELECT
SET H7.01  ; SENSOR SELECTED
RSET H7.00  ; SWITCH SELECTED

### Section MANUAL

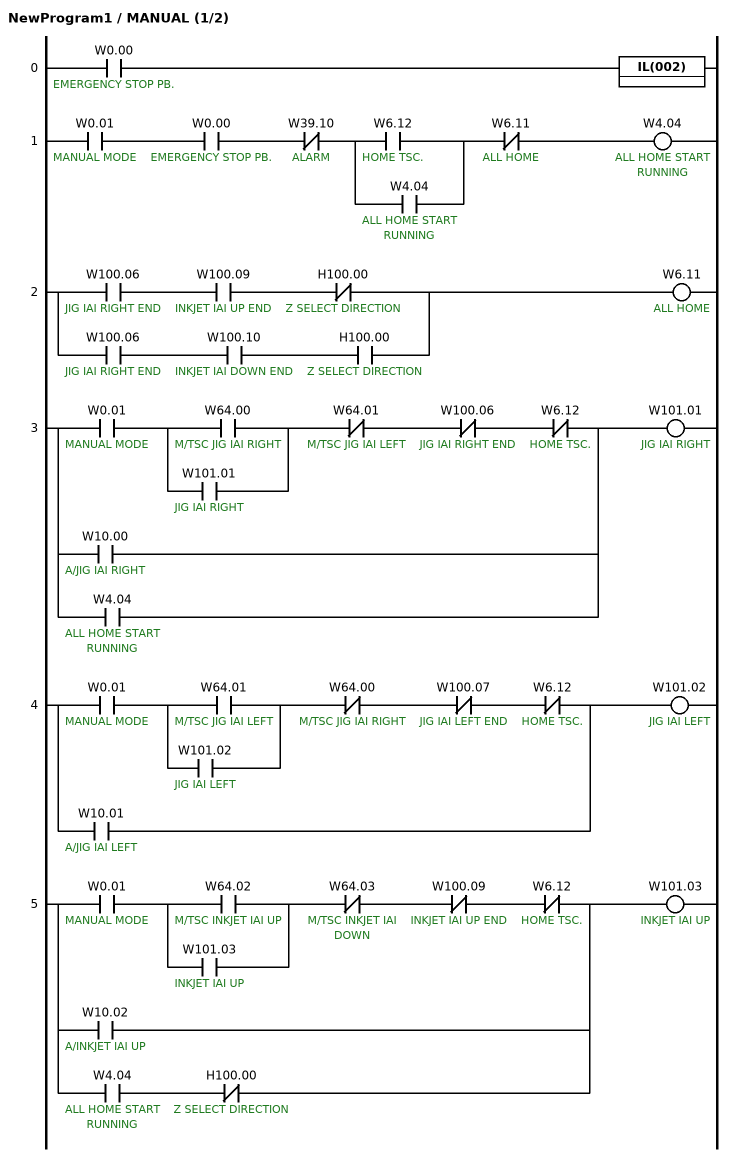
; rung 0
LD W0.00  ; EMERGENCY STOP PB.
IL(002)
; rung 1
LD W0.01  ; MANUAL MODE
AND W0.00  ; EMERGENCY STOP PB.
ANDNOT W39.10  ; ALARM
LD W6.12  ; HOME TSC.
OR W4.04  ; ALL HOME START RUNNING
ANDLD
ANDNOT W6.11  ; ALL HOME
OUT W4.04  ; ALL HOME START RUNNING
; rung 2
LD W100.06  ; JIG IAI RIGHT END
AND W100.09  ; INKJET IAI UP END
ANDNOT H100.00  ; Z SELECT DIRECTION
LD W100.06  ; JIG IAI RIGHT END
AND W100.10  ; INKJET IAI DOWN END
AND H100.00  ; Z SELECT DIRECTION
ORLD
OUT W6.11  ; ALL HOME
; rung 3
LD W0.01  ; MANUAL MODE
LD W64.00  ; M/TSC JIG IAI RIGHT
OR W101.01  ; JIG IAI RIGHT
ANDLD
ANDNOT W64.01  ; M/TSC JIG IAI LEFT
ANDNOT W100.06  ; JIG IAI RIGHT END
ANDNOT W6.12  ; HOME TSC.
LD W10.00  ; A/JIG IAI RIGHT
OR W4.04  ; ALL HOME START RUNNING
ORLD
OUT W101.01  ; JIG IAI RIGHT
; rung 4
LD W0.01  ; MANUAL MODE
LD W64.01  ; M/TSC JIG IAI LEFT
OR W101.02  ; JIG IAI LEFT
ANDLD
ANDNOT W64.00  ; M/TSC JIG IAI RIGHT
ANDNOT W100.07  ; JIG IAI LEFT END
ANDNOT W6.12  ; HOME TSC.
OR W10.01  ; A/JIG IAI LEFT
OUT W101.02  ; JIG IAI LEFT
; rung 5
LD W0.01  ; MANUAL MODE
LD W64.02  ; M/TSC INKJET IAI UP
OR W101.03  ; INKJET IAI UP
ANDLD
ANDNOT W64.03  ; M/TSC INKJET IAI DOWN
ANDNOT W100.09  ; INKJET IAI UP END
ANDNOT W6.12  ; HOME TSC.
OR W10.02  ; A/INKJET IAI UP
LD W4.04  ; ALL HOME START RUNNING
ANDNOT H100.00  ; Z SELECT DIRECTION
ORLD
OUT W101.03  ; INKJET IAI UP

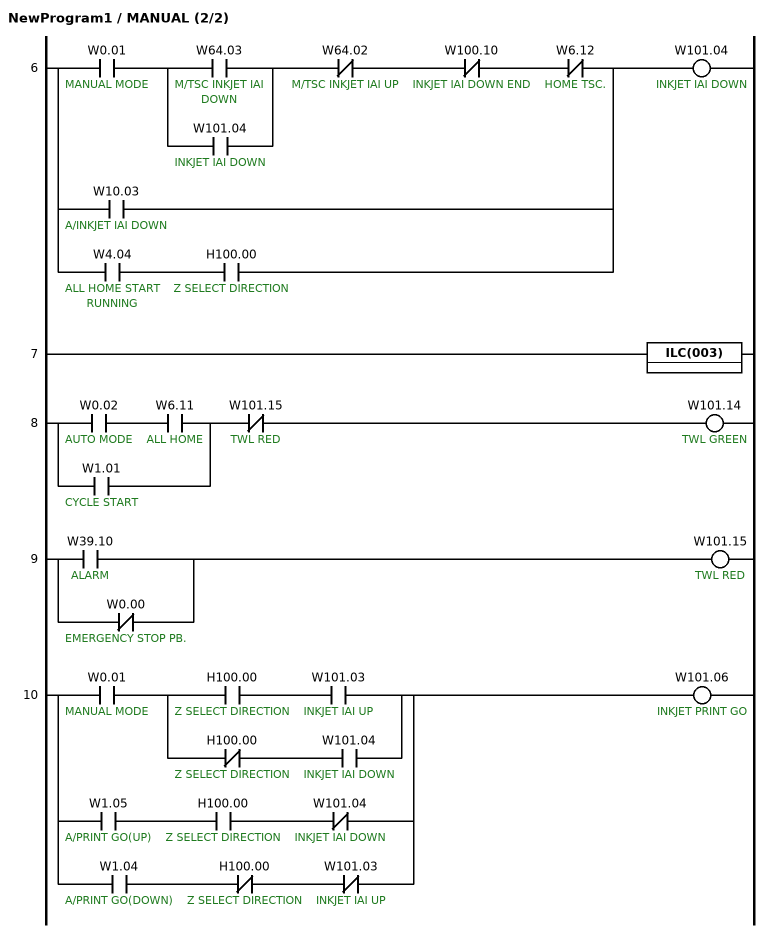
; rung 6
LD W0.01  ; MANUAL MODE
LD W64.03  ; M/TSC INKJET IAI DOWN
OR W101.04  ; INKJET IAI DOWN
ANDLD
ANDNOT W64.02  ; M/TSC INKJET IAI UP
ANDNOT W100.10  ; INKJET IAI DOWN END
ANDNOT W6.12  ; HOME TSC.
OR W10.03  ; A/INKJET IAI DOWN
LD W4.04  ; ALL HOME START RUNNING
AND H100.00  ; Z SELECT DIRECTION
ORLD
OUT W101.04  ; INKJET IAI DOWN
; rung 7
ILC(003)
; rung 8
LD W0.02  ; AUTO MODE
AND W6.11  ; ALL HOME
OR W1.01  ; CYCLE START
ANDNOT W101.15  ; TWL RED
OUT W101.14  ; TWL GREEN
; rung 9
LD W39.10  ; ALARM
ORNOT W0.00  ; EMERGENCY STOP PB.
OUT W101.15  ; TWL RED
; rung 10
LD W0.01  ; MANUAL MODE
LD H100.00  ; Z SELECT DIRECTION
AND W101.03  ; INKJET IAI UP
LDNOT H100.00  ; Z SELECT DIRECTION
AND W101.04  ; INKJET IAI DOWN
ORLD
ANDLD
LD W1.05  ; A/PRINT GO(UP)
AND H100.00  ; Z SELECT DIRECTION
ANDNOT W101.04  ; INKJET IAI DOWN
ORLD
LD W1.04  ; A/PRINT GO(DOWN)
ANDNOT H100.00  ; Z SELECT DIRECTION
ANDNOT W101.03  ; INKJET IAI UP
ORLD
OUT W101.06  ; INKJET PRINT GO

### Section INPUT

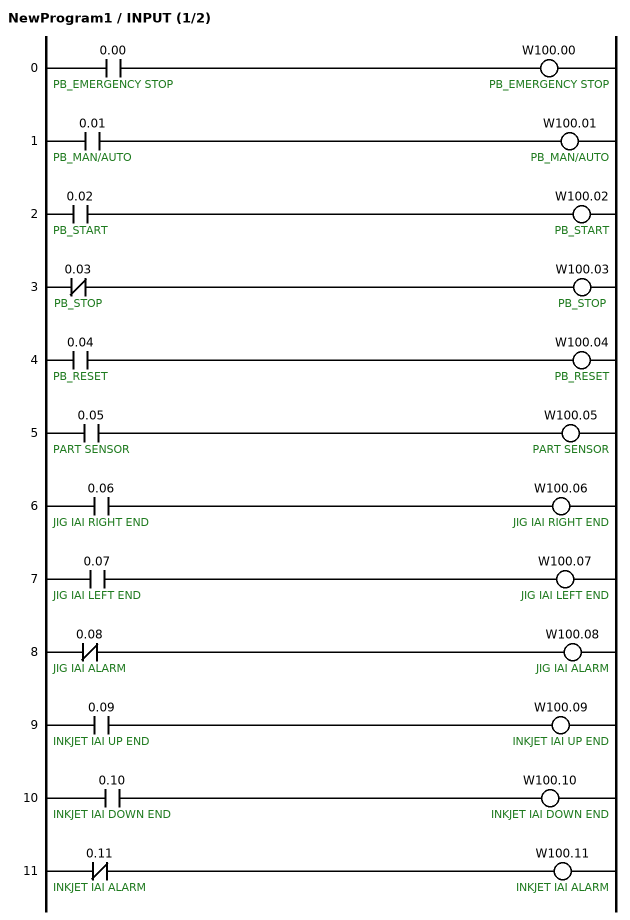
; rung 0
LD 0.00  ; PB_EMERGENCY STOP
OUT W100.00  ; PB_EMERGENCY STOP
; rung 1
LD 0.01  ; PB_MAN/AUTO
OUT W100.01  ; PB_MAN/AUTO
; rung 2
LD 0.02  ; PB_START
OUT W100.02  ; PB_START
; rung 3
LDNOT 0.03  ; PB_STOP
OUT W100.03  ; PB_STOP
; rung 4
LD 0.04  ; PB_RESET
OUT W100.04  ; PB_RESET
; rung 5
LD 0.05  ; PART SENSOR
OUT W100.05  ; PART SENSOR
; rung 6
LD 0.06  ; JIG IAI RIGHT END
OUT W100.06  ; JIG IAI RIGHT END
; rung 7
LD 0.07  ; JIG IAI LEFT END
OUT W100.07  ; JIG IAI LEFT END
; rung 8
LDNOT 0.08  ; JIG IAI ALARM
OUT W100.08  ; JIG IAI ALARM
; rung 9
LD 0.09  ; INKJET IAI UP END
OUT W100.09  ; INKJET IAI UP END
; rung 10
LD 0.10  ; INKJET IAI DOWN END
OUT W100.10  ; INKJET IAI DOWN END
; rung 11
LDNOT 0.11  ; INKJET IAI ALARM
OUT W100.11  ; INKJET IAI ALARM

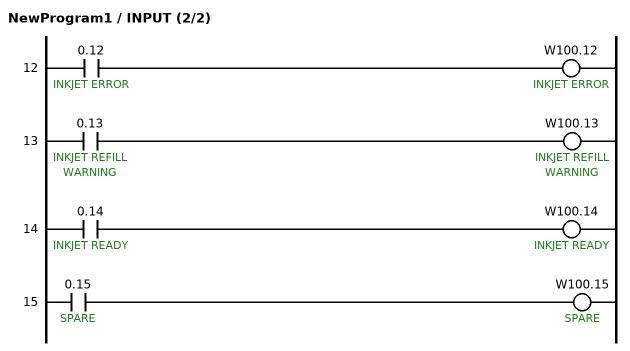
; rung 12
LD 0.12  ; INKJET ERROR
OUT W100.12  ; INKJET ERROR
; rung 13
LD 0.13  ; INKJET REFILL WARNING
OUT W100.13  ; INKJET REFILL WARNING
; rung 14
LD 0.14  ; INKJET READY
OUT W100.14  ; INKJET READY
; rung 15
LD 0.15  ; SPARE
OUT W100.15  ; SPARE

### Section OUTPUT

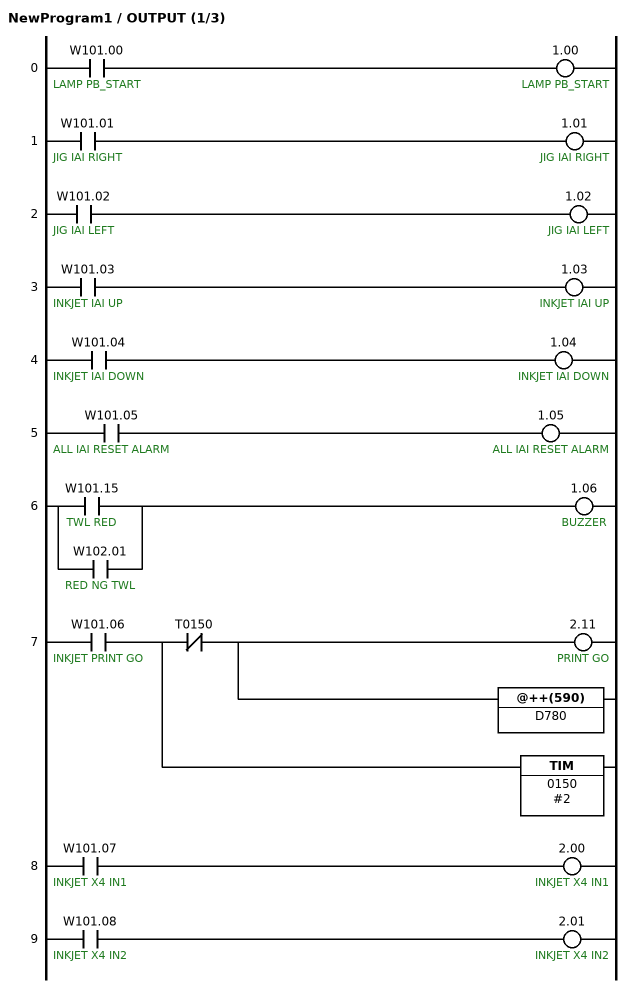
; rung 0
LD W101.00  ; LAMP PB_START
OUT 1.00  ; LAMP PB_START
; rung 1
LD W101.01  ; JIG IAI RIGHT
OUT 1.01  ; JIG IAI RIGHT
; rung 2
LD W101.02  ; JIG IAI LEFT
OUT 1.02  ; JIG IAI LEFT
; rung 3
LD W101.03  ; INKJET IAI UP
OUT 1.03  ; INKJET IAI UP
; rung 4
LD W101.04  ; INKJET IAI DOWN
OUT 1.04  ; INKJET IAI DOWN
; rung 5
LD W101.05  ; ALL IAI RESET ALARM
OUT 1.05  ; ALL IAI RESET ALARM
; rung 6
LD W101.15  ; TWL RED
OR W102.01  ; RED NG TWL
OUT 1.06  ; BUZZER
; rung 7
LD W101.06  ; INKJET PRINT GO
OUT TR0
ANDNOT T0150
OUT 2.11  ; PRINT GO
@++(590) D780
LD TR0
TIM 0150 #2
; rung 8
LD W101.07  ; INKJET X4 IN1
OUT 2.00  ; INKJET X4 IN1
; rung 9
LD W101.08  ; INKJET X4 IN2
OUT 2.01  ; INKJET X4 IN2

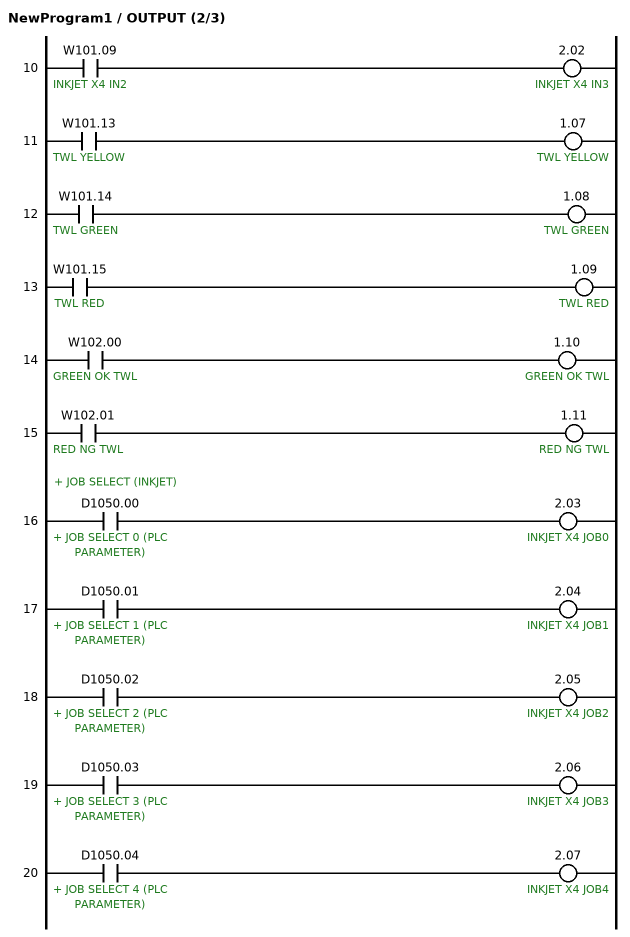
; rung 10
LD W101.09  ; INKJET X4 IN2
OUT 2.02  ; INKJET X4 IN3
; rung 11
LD W101.13  ; TWL YELLOW
OUT 1.07  ; TWL YELLOW
; rung 12
LD W101.14  ; TWL GREEN
OUT 1.08  ; TWL GREEN
; rung 13
LD W101.15  ; TWL RED
OUT 1.09  ; TWL RED
; rung 14
LD W102.00  ; GREEN OK TWL
OUT 1.10  ; GREEN OK TWL
; rung 15
LD W102.01  ; RED NG TWL
OUT 1.11  ; RED NG TWL
; rung 16: + JOB SELECT (INKJET)
LD D1050.00  ; + JOB SELECT 0 (PLC PARAMETER)
OUT 2.03  ; INKJET X4 JOB0
; rung 17
LD D1050.01  ; + JOB SELECT 1 (PLC PARAMETER)
OUT 2.04  ; INKJET X4 JOB1
; rung 18
LD D1050.02  ; + JOB SELECT 2 (PLC PARAMETER)
OUT 2.05  ; INKJET X4 JOB2
; rung 19
LD D1050.03  ; + JOB SELECT 3 (PLC PARAMETER)
OUT 2.06  ; INKJET X4 JOB3
; rung 20
LD D1050.04  ; + JOB SELECT 4 (PLC PARAMETER)
OUT 2.07  ; INKJET X4 JOB4

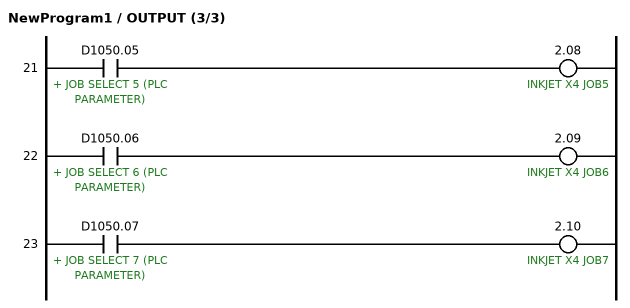
; rung 21
LD D1050.05  ; + JOB SELECT 5 (PLC PARAMETER)
OUT 2.08  ; INKJET X4 JOB5
; rung 22
LD D1050.06  ; + JOB SELECT 6 (PLC PARAMETER)
OUT 2.09  ; INKJET X4 JOB6
; rung 23
LD D1050.07  ; + JOB SELECT 7 (PLC PARAMETER)
OUT 2.10  ; INKJET X4 JOB7

### Section ALARM

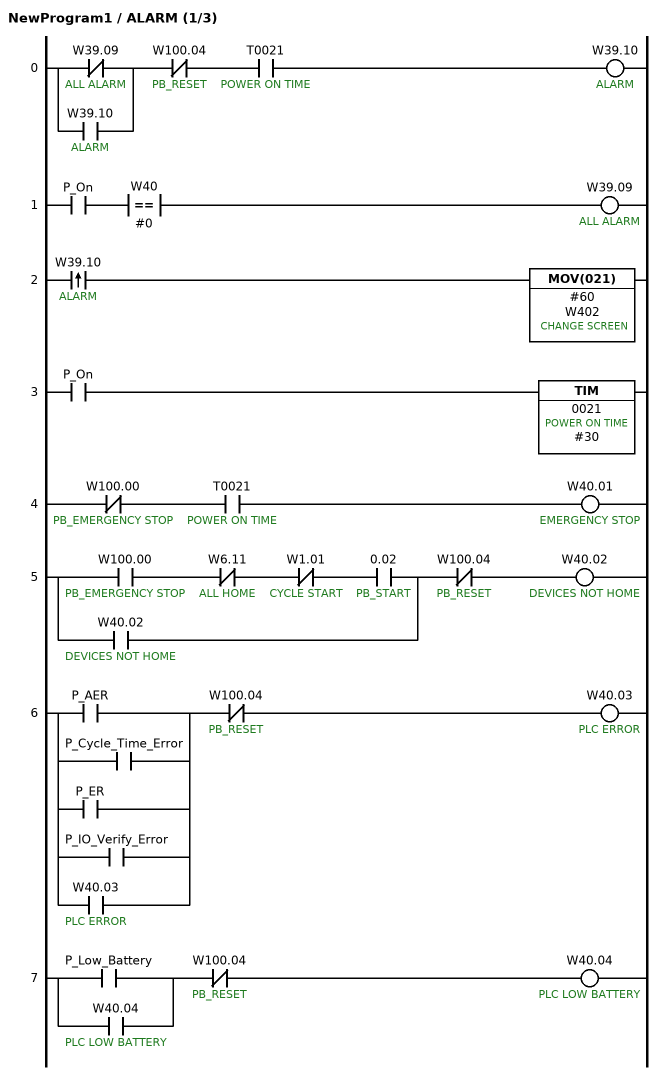
; rung 0
LDNOT W39.09  ; ALL ALARM
OR W39.10  ; ALARM
ANDNOT W100.04  ; PB_RESET
AND T0021  ; POWER ON TIME
OUT W39.10  ; ALARM
; rung 1
LD P_On
AND=(300) W40 #0
OUT W39.09  ; ALL ALARM
; rung 2
@LD W39.10  ; ALARM
MOV(021) #60 W402  ; CHANGE SCREEN
; rung 3
LD P_On
TIM 0021 #30  ; POWER ON TIME
; rung 4
LDNOT W100.00  ; PB_EMERGENCY STOP
AND T0021  ; POWER ON TIME
OUT W40.01  ; EMERGENCY STOP
; rung 5
LD W100.00  ; PB_EMERGENCY STOP
ANDNOT W6.11  ; ALL HOME
ANDNOT W1.01  ; CYCLE START
AND 0.02  ; PB_START
OR W40.02  ; DEVICES NOT HOME
ANDNOT W100.04  ; PB_RESET
OUT W40.02  ; DEVICES NOT HOME
; rung 6
LD P_AER
OR P_Cycle_Time_Error
OR P_ER
OR P_IO_Verify_Error
OR W40.03  ; PLC ERROR
ANDNOT W100.04  ; PB_RESET
OUT W40.03  ; PLC ERROR
; rung 7
LD P_Low_Battery
OR W40.04  ; PLC LOW BATTERY
ANDNOT W100.04  ; PB_RESET
OUT W40.04  ; PLC LOW BATTERY

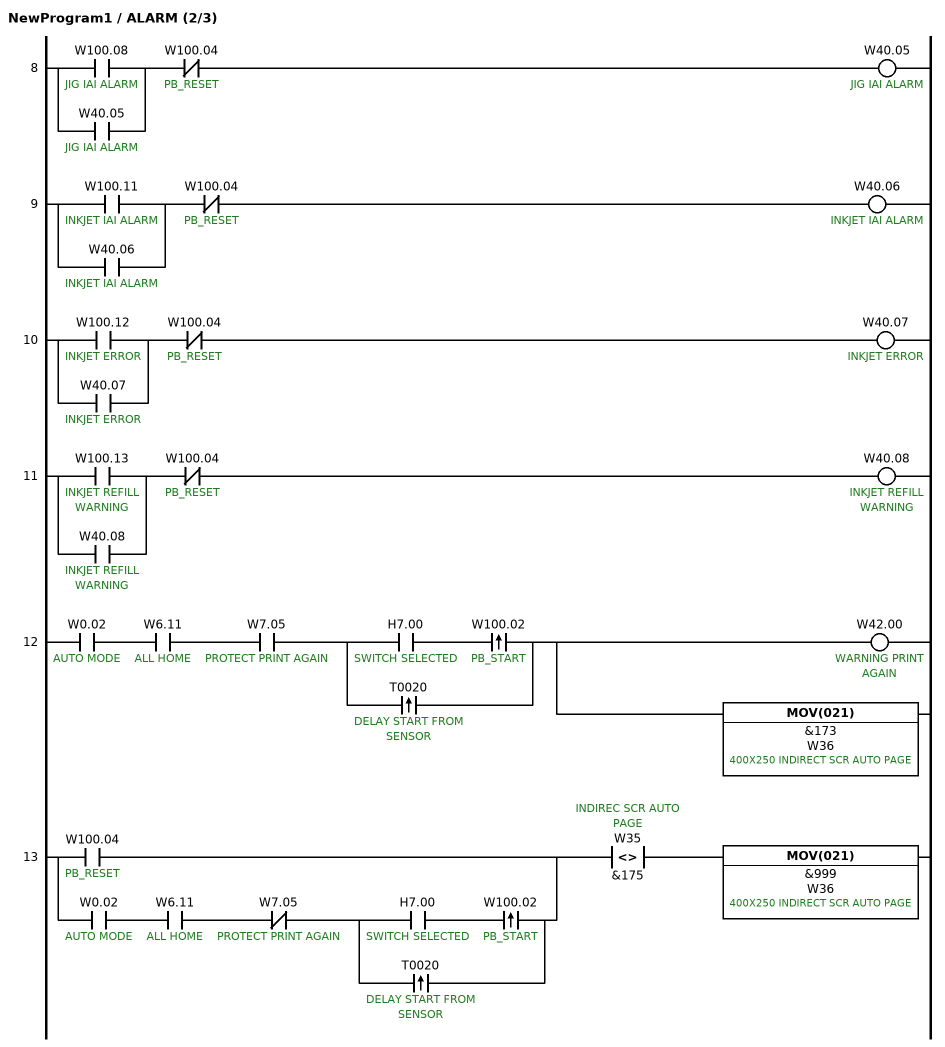
; rung 8
LD W100.08  ; JIG IAI ALARM
OR W40.05  ; JIG IAI ALARM
ANDNOT W100.04  ; PB_RESET
OUT W40.05  ; JIG IAI ALARM
; rung 9
LD W100.11  ; INKJET IAI ALARM
OR W40.06  ; INKJET IAI ALARM
ANDNOT W100.04  ; PB_RESET
OUT W40.06  ; INKJET IAI ALARM
; rung 10
LD W100.12  ; INKJET ERROR
OR W40.07  ; INKJET ERROR
ANDNOT W100.04  ; PB_RESET
OUT W40.07  ; INKJET ERROR
; rung 11
LD W100.13  ; INKJET REFILL WARNING
OR W40.08  ; INKJET REFILL WARNING
ANDNOT W100.04  ; PB_RESET
OUT W40.08  ; INKJET REFILL WARNING
; rung 12
LD W0.02  ; AUTO MODE
AND W6.11  ; ALL HOME
AND W7.05  ; PROTECT PRINT AGAIN
LD H7.00  ; SWITCH SELECTED
@AND W100.02  ; PB_START
@OR T0020  ; DELAY START FROM SENSOR
ANDLD
OUT W42.00  ; WARNING PRINT AGAIN
MOV(021) &173 W36  ; 400X250 INDIRECT SCR AUTO PAGE
; rung 13
LD W100.04  ; PB_RESET
LD W0.02  ; AUTO MODE
AND W6.11  ; ALL HOME
ANDNOT W7.05  ; PROTECT PRINT AGAIN
LD H7.00  ; SWITCH SELECTED
@AND W100.02  ; PB_START
@OR T0020  ; DELAY START FROM SENSOR
ANDLD
ORLD
AND<>(305) W35 &175  ; INDIREC SCR AUTO PAGE
MOV(021) &999 W36  ; 400X250 INDIRECT SCR AUTO PAGE

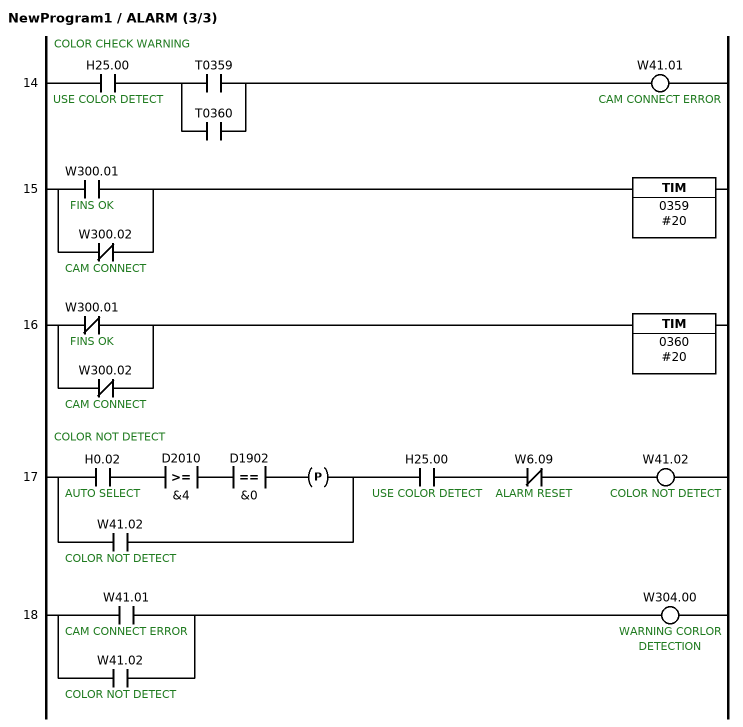
; rung 14: COLOR CHECK WARNING
LD H25.00  ; USE COLOR DETECT
LD T0359
OR T0360
ANDLD
OUT W41.01  ; CAM CONNECT ERROR
; rung 15
LD W300.01  ; FINS OK
ORNOT W300.02  ; CAM CONNECT
TIM 0359 #20
; rung 16
LDNOT W300.01  ; FINS OK
ORNOT W300.02  ; CAM CONNECT
TIM 0360 #20
; rung 17: COLOR NOT DETECT
LD H0.02  ; AUTO SELECT
AND>=(325) D2010 &4
AND=L(301) D1902 &0
UP(521)
OR W41.02  ; COLOR NOT DETECT
AND H25.00  ; USE COLOR DETECT
ANDNOT W6.09  ; ALARM RESET
OUT W41.02  ; COLOR NOT DETECT
; rung 18
LD W41.01  ; CAM CONNECT ERROR
OR W41.02  ; COLOR NOT DETECT
OUT W304.00  ; WARNING CORLOR DETECTION

### Section BARCODE

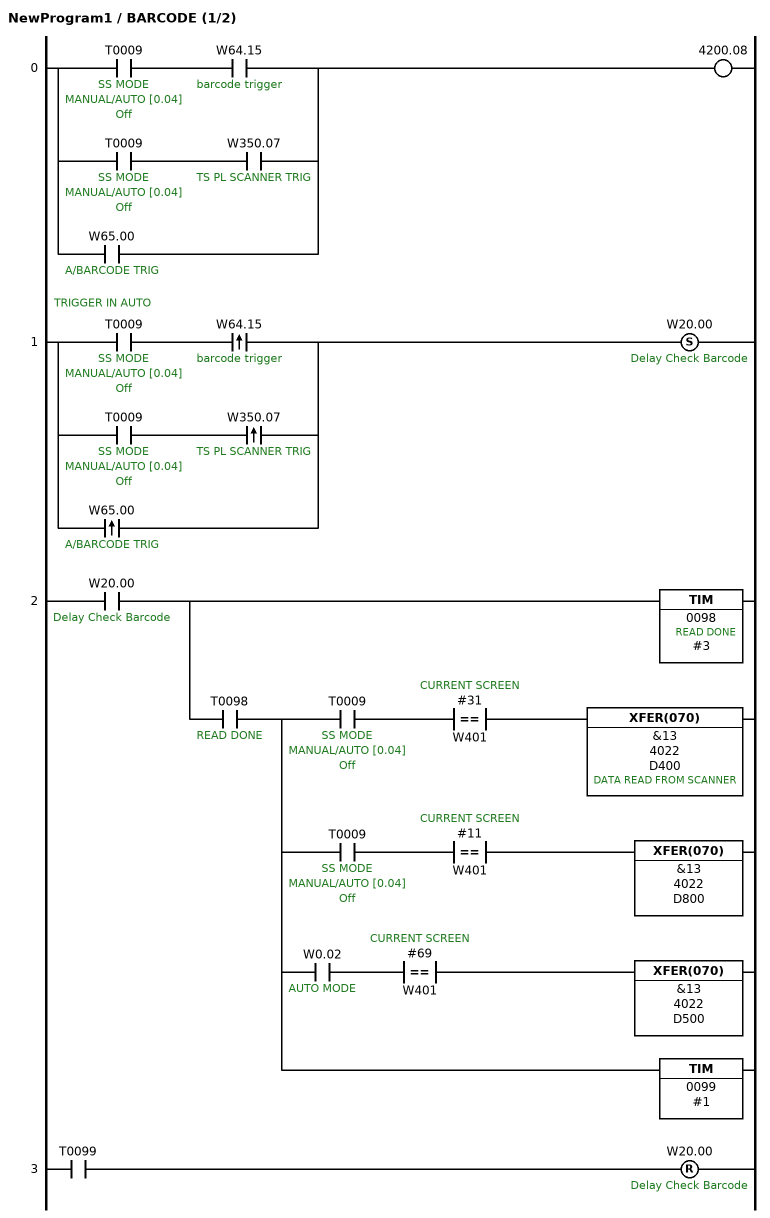
; rung 0
LD T0009  ; SS MODE MANUAL/AUTO [0.04] Off
AND W64.15  ; barcode trigger
LD T0009  ; SS MODE MANUAL/AUTO [0.04] Off
AND W350.07  ; TS PL SCANNER TRIG
ORLD
OR W65.00  ; A/BARCODE TRIG
OUT 4200.08
; rung 1: TRIGGER IN AUTO
LD T0009  ; SS MODE MANUAL/AUTO [0.04] Off
@AND W64.15  ; barcode trigger
LD T0009  ; SS MODE MANUAL/AUTO [0.04] Off
@AND W350.07  ; TS PL SCANNER TRIG
ORLD
@OR W65.00  ; A/BARCODE TRIG
SET W20.00  ; Delay Check Barcode
; rung 2
LD W20.00  ; Delay Check Barcode
TIM 0098 #3  ; READ DONE
AND T0098  ; READ DONE
OUT TR0
AND T0009  ; SS MODE MANUAL/AUTO [0.04] Off
AND=(300) #31 W401  ; CURRENT SCREEN
XFER(070) &13 4022 D400  ; DATA READ FROM SCANNER
LD TR0
AND T0009  ; SS MODE MANUAL/AUTO [0.04] Off
AND=(300) #11 W401  ; CURRENT SCREEN
XFER(070) &13 4022 D800
LD TR0
AND W0.02  ; AUTO MODE
AND=(300) #69 W401  ; CURRENT SCREEN
XFER(070) &13 4022 D500
LD TR0
TIM 0099 #1
; rung 3
LD T0099
RSET W20.00  ; Delay Check Barcode

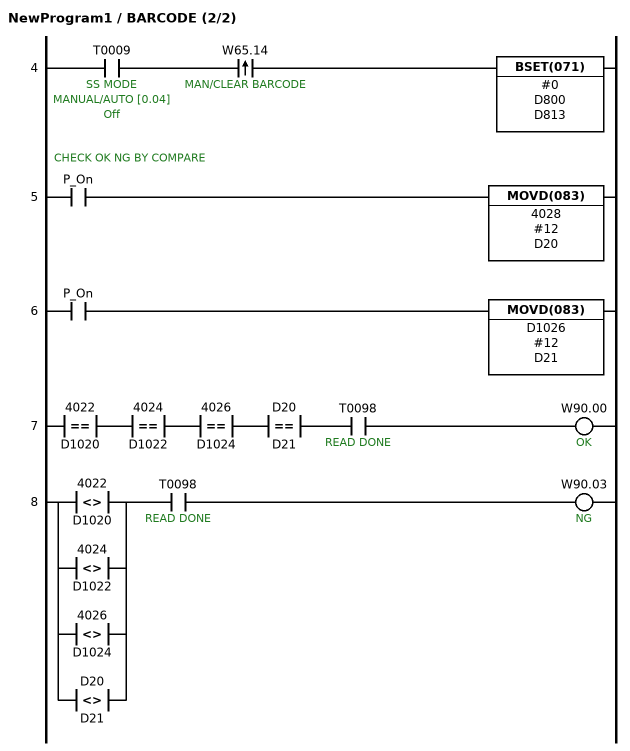
; rung 4
LD T0009  ; SS MODE MANUAL/AUTO [0.04] Off
@AND W65.14  ; MAN/CLEAR BARCODE
BSET(071) #0 D800 D813
; rung 5: CHECK OK NG BY COMPARE
LD P_On
MOVD(083) 4028 #12 D20
; rung 6
LD P_On
MOVD(083) D1026 #12 D21
; rung 7
LD=L(301) 4022 D1020
AND=L(301) 4024 D1022
AND=L(301) 4026 D1024
AND=(300) D20 D21
AND T0098  ; READ DONE
OUT W90.00  ; OK
; rung 8
LD<>L(306) 4022 D1020
OR<>L(306) 4024 D1022
OR<>L(306) 4026 D1024
OR<>(305) D20 D21
AND T0098  ; READ DONE
OUT W90.03  ; NG

### Section SCANNER

